{attribute 'linkalways'} 
{attribute 'no_explicit_call' := 'This FB is a CLASS and must be accessed using methods or properties'}
{attribute 'enable_dynamic_creation'}
FUNCTION_BLOCK _ETcVnOrientationMethod EXTENDS EnumDatatypeBase
VAR
	localData : ETcVnOrientationMethod;
	activeData : REFERENCE TO ETcVnOrientationMethod;
	enumBaseDatatype : _DINT(localData);
END_VAR

METHOD PRIVATE AddLocalEnumeration
VAR_INPUT
	Enumeration : T_MAXSTRING;
	Value : ETcVnOrientationMethod;
END_VAR
AddEnumeration(Enumeration, Value);
END_METHOD

PROPERTY PUBLIC Address : PVOID
GET
Address := ADR(activeData);
END_GET
END_PROPERTY

METHOD PUBLIC ClearReference
VAR_INPUT
END_VAR
activeData REF= localData;
SetBaseDatatypeReference();
END_METHOD

METHOD PUBLIC Clone : I_Datatype
VAR
    pClone : POINTER TO _ETcVnOrientationMethod;
END_VAR
pClone := __NEW(_ETcVnOrientationMethod(InitialValue := Value));
Clone := pClone^;
END_METHOD

METHOD FB_init : BOOL
VAR_INPUT
	bInitRetains : BOOL; // if TRUE, the retain variables are initialized (warm start / cold start)
	bInCopyCode : BOOL;  // if TRUE, the instance afterwards gets moved into the copy code (online change)
	InitialValue : ETcVnOrientationMethod;
END_VAR
localData := InitialValue;
AddBaseDatatype(enumBaseDatatype);
ClearReference();

AddLocalEnumeration('TCVN_OM_PCA', ETcVnOrientationMethod.TCVN_OM_PCA);
AddLocalEnumeration('TCVN_OM_FITELLIPSE', ETcVnOrientationMethod.TCVN_OM_FITELLIPSE);
AddLocalEnumeration('TCVN_OM_MOMENTS', ETcVnOrientationMethod.TCVN_OM_MOMENTS);
AddLocalEnumeration('TCVN_OM_ENCLOSINGRECT', ETcVnOrientationMethod.TCVN_OM_ENCLOSINGRECT);
END_METHOD

PROPERTY PUBLIC Identifier : T_MAXSTRING
GET
Identifier := 'ETcVnOrientationMethod';
END_GET
END_PROPERTY

METHOD IsEnumeratorValueEqual : BOOL
VAR_INPUT
	Enumerator : I_KeyValueForwardEnumerator;
END_VAR
VAR
	storedValue : ETcVnOrientationMethod;
END_VAR
IF NOT Enumerator.TryGet(storedValue) THEN
	RETURN;
END_IF

IsEnumeratorValueEqual := storedValue = activeData;
END_METHOD

METHOD PUBLIC MakeReferenceTo
VAR_INPUT
	ReferenceTarget : REFERENCE TO ETcVnOrientationMethod;
END_VAR
activeData REF= ReferenceTarget;
SetBaseDatatypeReference();
END_METHOD

METHOD PROTECTED SetBaseDatatypeReference
VAR_INPUT
END_VAR
enumBaseDatatype.MakeReferenceTo(activeData);
END_METHOD

PROPERTY PUBLIC Size : UDINT
GET
Size := SIZEOF(activeData);
END_GET
END_PROPERTY

METHOD TryMakeReferenceTo : BOOL
VAR_INPUT
	Target : I_Datatype;
END_VAR
VAR
	targetAsEnum : I_EnumDatatype;
	pTargetData : POINTER TO ETcVnOrientationMethod;
END_VAR
IF NOT Target.TryResolveAsEnumDatatype(targetAsEnum) THEN
	RETURN;
END_IF

IF targetAsEnum.Identifier <> Identifier THEN
	RETURN;
END_IF

pTargetData := Target.Address;
activeData REF= pTargetData^;
SetBaseDatatypeReference();
TryMakeReferenceTo := TRUE;
END_METHOD

PROPERTY PUBLIC Value : ETcVnOrientationMethod
GET
Value := activeData;
END_GET
SET
activeData := Value;
END_SET
END_PROPERTY

END_FUNCTION_BLOCK

(* stored: Version 1.1.0.1, ProductVersion 3.1.4024.12
   POU _ETcVnOrientationMethod: Id {97bdb7bd-41a7-43dd-beee-51af0176e725}, SpecialFunc None
   Folder Constructor: Id {7049d346-f6b1-4797-83d8-6ffd08e40c80}
   Folder Private: Id {c2617cde-4ac8-493f-92b7-5b0c0a9d8595}
   Folder Protected: Id {4fdc26a1-1d18-44c7-889b-da966ddf7c1e}
   Method AddLocalEnumeration: Id {5fce8bdd-10ec-41c5-b44a-8b00e07311f5}
   Property Address: Id {d243987a-3955-46fd-9319-56ed48b3cc57}
   Get Get: Id {d1c4564a-8861-4c36-a573-98d6229723f6}
   Method ClearReference: Id {5a9d6c1c-d4d8-4a55-9510-52393d22a558}
   Method Clone: Id {613e5fa3-8a63-42d6-b733-971e6457195a}
   Method FB_init: Id {bb391d47-f440-419f-a746-9d2a3c1b93f8}
   Property Identifier: Id {3e10f703-8451-4b73-b579-5b7930d4d2c4}
   Get Get: Id {42361a53-5c02-486f-b91c-6d2edeb31761}
   Method IsEnumeratorValueEqual: Id {c40d83b6-3f86-4b18-a9a4-5f9c0f7b8ffd}
   Method MakeReferenceTo: Id {ab92bbcc-bd6f-4778-86f7-921334ab8d43}
   Method SetBaseDatatypeReference: Id {b91e44f6-14f1-4d15-a765-458abda28602}
   Property Size: Id {d932337e-b5c2-4d4e-beca-d29673b2f0d3}
   Get Get: Id {870be4e9-d703-41d1-9982-b0e1ee30524d}
   Method TryMakeReferenceTo: Id {c98344ce-5a61-4952-a3c4-070596b1d9de}
   Property Value: Id {8773c8bf-ec24-4002-8dc4-2430634fec83}
   Get Get: Id {98d73d07-8323-4afb-8930-a2cf3ff81835}
   Set Set: Id {e099a674-6697-43f2-af55-570fca0aabc0} *)
